(* Logix 5000 project; controller HP_SSC01 vendor 1 type 14 code 67 rev 17.7; software revision 17.01; part 10 of 15 *)
(* tags used below, declared in another part *)
   A_C3_0422 : ALIAS FOR C3_Warning.22;
   A_C3_0423 : ALIAS FOR C3_Warning.23;
   A_C3_0425 : ALIAS FOR C3_Warning.25;
   A_C3_0426 : ALIAS FOR C3_Warning.26;
   C3 : AXIS_SERVO_DRIVE;
   C3_32HourTimers : TIMER[4];
   C3_ActualPositionMOD60 : REAL;
   C3_All_DLY_OK : BOOL;
   C3_Brake_Daily_ok : BOOL;
   C3_Brake_Test_passed : BOOL;
   C3_BrakeReleaseSelected : BOOL;
   C3_BrakeTestExpireTime : DINT;
   C3_BrakeTestExpireTimeTemp : DINT;
   C3_BrakeTestFailed : BOOL;
   C3_BrakeTestMessageNumber : DINT;
   C3_BrakeTestSelected : BOOL;
   C3_BrakeTestSequence : DINT;
   C3_BrakeTestWarning : BOOL;
   C3_DistanceToEvac : REAL;
   C3_Dump_OK : BOOL;
   C3_DumpValveReleaseSelected : BOOL;
   C3_DumpValveTestExpireTime : DINT;
   C3_DumpValveTestExpireTimeTemp : DINT;
   C3_DumpValveTestSelected : BOOL;
   C3_DumpValveTestSequence : DINT;
   C3_EvacPosition : REAL;
   C3_EvacPositionMOD60 : REAL;
   C3_ExcecutePBHoldTimer : TIMER;
   C3_FaultStandard : DINT;
   C3_GoNearOnPathDelay : TIMER;
   C3_GoToEvacMAM01 : MOTION_INSTRUCTION;
   C3_GoToOnPathMAM01 : MOTION_INSTRUCTION;
   C3_GoToOnPathMAM02 : MOTION_INSTRUCTION;
   C3_Home_OK : BOOL;
   C3_Homed : BOOL;
   C3_HomeExpireTime : DINT;
   C3_HomeExpireTimeTemp : DINT;
   C3_HomeSequence : DINT;
   C3_JogForwardFastSelected : BOOL;
   C3_JogForwardSlowSelected : BOOL;
   C3_JogReverseFastSelected : BOOL;
   C3_JogReverseSlowSelected : BOOL;
   C3_LubricationMessageNumber : DINT;
   C3_LubricationOnTimer : TIMER;
   C3_LubricationOverrideSelected : BOOL;
   C3_MAFR : MOTION_INSTRUCTION;
   C3_MAG : MOTION_INSTRUCTION;
   C3_MAJDeceleration : REAL;
   C3_MAS : MOTION_INSTRUCTION;
   C3_MASR : MOTION_INSTRUCTION;
   C3_Oiler : ALIAS FOR C3_RIO_AENT:O.Data[2].1;
   C3_OIT_BrakeRelease : BOOL;
   C3_OIT_BrakeReleaseDisplay : BOOL;
   C3_OIT_BrakeTest : BOOL;
   C3_OIT_BrakeTestDisplay : BOOL;
   C3_OIT_Command : DINT;
   C3_OIT_Current : DINT;
   C3_OIT_DumpValveRelease : BOOL;
   C3_OIT_DumpValveReleaseDisplay : BOOL;
   C3_OIT_DumpValveTest : BOOL;
   C3_OIT_DumpValveTestDisplay : BOOL;
   C3_OIT_FaultsExist : BOOL;
   C3_OIT_HomeCountDown : DINT;
   C3_OIT_JogForwardFast : BOOL;
   C3_OIT_JogForwardFastDisplay : BOOL;
   C3_OIT_JogForwardSlow : BOOL;
   C3_OIT_JogForwardSlowDisplay : BOOL;
   C3_OIT_JogReverseFast : BOOL;
   C3_OIT_JogReverseFastDisplay : BOOL;
   C3_OIT_JogReverseSlow : BOOL;
   C3_OIT_JogReverseSlowDisplay : BOOL;
   C3_OIT_JogStopDisplay : BOOL;
   C3_OIT_LubricationOverride : BOOL;
   C3_OIT_LubricationOverrideDisplay : BOOL;
   C3_OIT_PathError : DINT;
   C3_OIT_PathIndicatorHigh : DINT;
   C3_OIT_PathIndicatorLow : DINT;
   C3_OIT_WarningsExist : BOOL;
   C3_OneTryToFixErrorONS : BOOL;
   C3_ONS : DINT;
   C3_RemoteBrakeAndHomeSequence : DINT;
   C3_RemoteBrakeAndHomeSequenceAlarms : DINT;
   C3_RemoteBrakeAndHomeSequenceAlarmTimer : TIMER[8];
   C3_RemoteBrakeAndHomeSequenceONS : BOOL;
   C3_RemoteBrakeTestCMD : BOOL;
   C3_RemoteDumpTestCMD : BOOL;
   C3_RemoteHomeCMD : BOOL;
   C3_RemoteScreenMessageNumber : DINT;
   C3_RemoteSequenceDelay : TIMER[4];
   C3_RevolutionCounter : COUNTER;
   C3_ServoActionStatusOnDelay : TIMER;
   C3_TargetPositionError : REAL;
   C3_TargetPositionErrorTest : REAL;
   C3_Warning : DINT;
   MasterClockCopyMAS_Stop1 : MOTION_INSTRUCTION;
   MasterClockCopyMAS_Stop2 : MOTION_INSTRUCTION;
   MasterClockLocal : AXIS_VIRTUAL;
   RCS_CMD_Auto_TON : TIMER;
   RCS_MasterClockLocalTagetDegrees : REAL;
   S_C3_FaultReset : BOOL;
   S_C3_FaultSafety : DINT;
   S_C3_ModeLocal : BOOL;
   S_C3_ModeRemote : BOOL;
   S_C3_MSTOP_InputOK : BOOL;
   S_C3_NearOnPath : BOOL;
   S_C3_NearOnPathHi : DINT;
   S_C3_NearOnPathLow : DINT;
   S_C3_OffPath : BOOL;
   S_C3_OnPath : BOOL;
   S_C3_PathError : DINT;
   S_RCS_MotionCMD_BrakeTest : BOOL;
   S_RCS_MotionCMD_Evac : BOOL;
   S_RCS_MotionCMD_GoNearOnPath : BOOL;
(* Carousel3, continued *)

ROUTINE C345_Lubrication   (* ladder *)
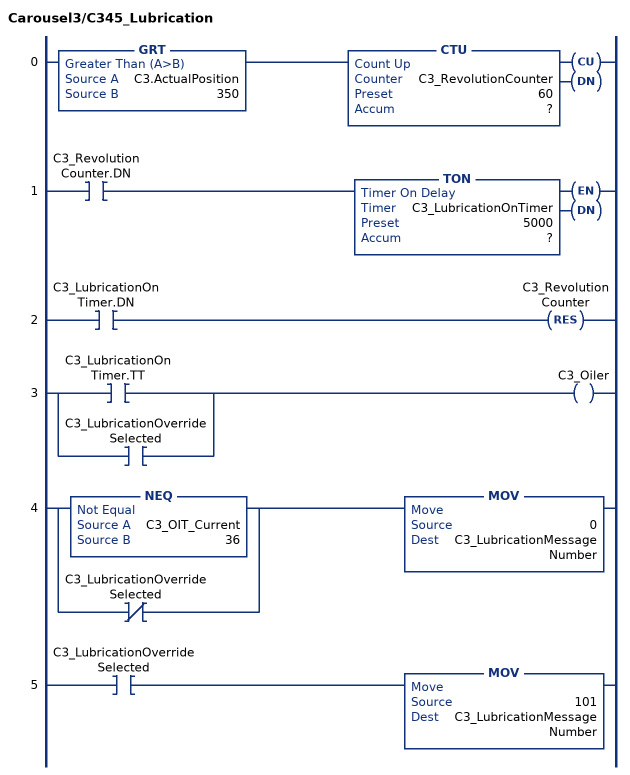
   0: GRT(C3.ActualPosition,350)CTU(C3_RevolutionCounter,?,?);
   1: XIC(C3_RevolutionCounter.DN)TON(C3_LubricationOnTimer,?,?);
   2: XIC(C3_LubricationOnTimer.DN)RES(C3_RevolutionCounter);
   3: [XIC(C3_LubricationOnTimer.TT) ,XIC(C3_LubricationOverrideSelected) ]OTE(C3_Oiler);
   4: [NEQ(C3_OIT_Current,36) ,XIO(C3_LubricationOverrideSelected) ]MOV(0,C3_LubricationMessageNumber);
   5: XIC(C3_LubricationOverrideSelected)MOV(101,C3_LubricationMessageNumber);
END_ROUTINE

ROUTINE C350_OIT   (* ladder *)
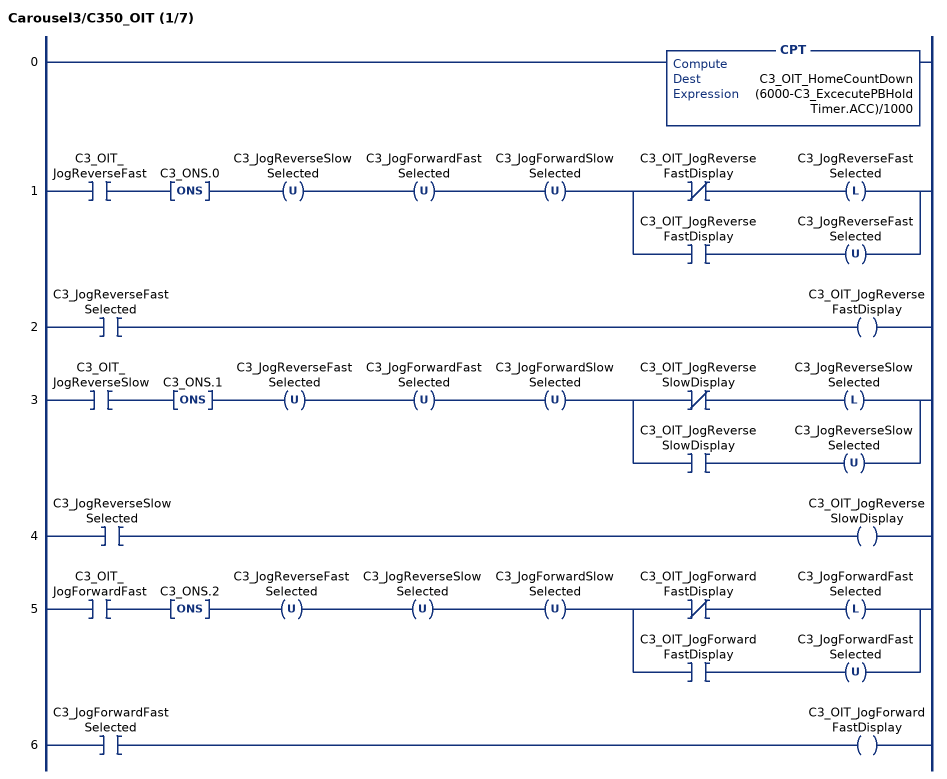
   0: CPT(C3_OIT_HomeCountDown,(6000-C3_ExcecutePBHoldTimer.ACC)/1000);
   1: XIC(C3_OIT_JogReverseFast)ONS(C3_ONS.0)OTU(C3_JogReverseSlowSelected)OTU(C3_JogForwardFastSelected)OTU(C3_JogForwardSlowSelected)[XIO(C3_OIT_JogReverseFastDisplay) OTL(C3_JogReverseFastSelected) ,XIC(C3_OIT_JogReverseFastDisplay) OTU(C3_JogReverseFastSelected) ];
   2: XIC(C3_JogReverseFastSelected)OTE(C3_OIT_JogReverseFastDisplay);
   3: XIC(C3_OIT_JogReverseSlow)ONS(C3_ONS.1)OTU(C3_JogReverseFastSelected)OTU(C3_JogForwardFastSelected)OTU(C3_JogForwardSlowSelected)[XIO(C3_OIT_JogReverseSlowDisplay) OTL(C3_JogReverseSlowSelected) ,XIC(C3_OIT_JogReverseSlowDisplay) OTU(C3_JogReverseSlowSelected) ];
   4: XIC(C3_JogReverseSlowSelected)OTE(C3_OIT_JogReverseSlowDisplay);
   5: XIC(C3_OIT_JogForwardFast)ONS(C3_ONS.2)OTU(C3_JogReverseFastSelected)OTU(C3_JogReverseSlowSelected)OTU(C3_JogForwardSlowSelected)[XIO(C3_OIT_JogForwardFastDisplay) OTL(C3_JogForwardFastSelected) ,XIC(C3_OIT_JogForwardFastDisplay) OTU(C3_JogForwardFastSelected) ];
   6: XIC(C3_JogForwardFastSelected)OTE(C3_OIT_JogForwardFastDisplay);
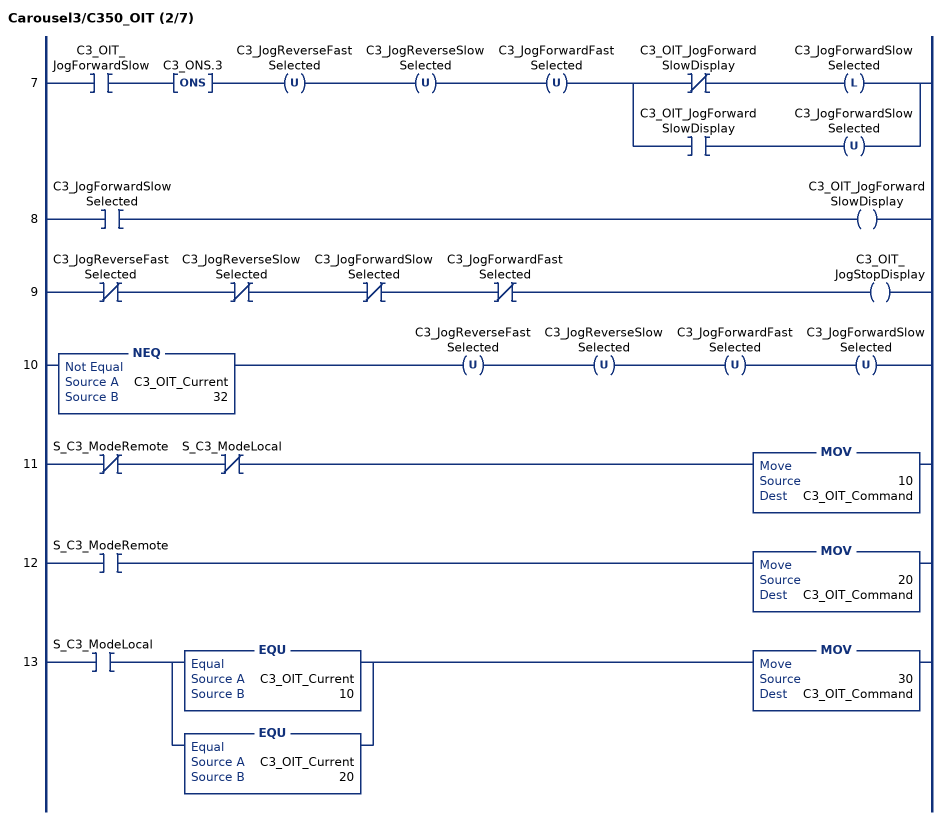
   7: XIC(C3_OIT_JogForwardSlow)ONS(C3_ONS.3)OTU(C3_JogReverseFastSelected)OTU(C3_JogReverseSlowSelected)OTU(C3_JogForwardFastSelected)[XIO(C3_OIT_JogForwardSlowDisplay) OTL(C3_JogForwardSlowSelected) ,XIC(C3_OIT_JogForwardSlowDisplay) OTU(C3_JogForwardSlowSelected) ];
   8: XIC(C3_JogForwardSlowSelected)OTE(C3_OIT_JogForwardSlowDisplay);
   9: XIO(C3_JogReverseFastSelected)XIO(C3_JogReverseSlowSelected)XIO(C3_JogForwardSlowSelected)XIO(C3_JogForwardFastSelected)OTE(C3_OIT_JogStopDisplay);
   10: NEQ(C3_OIT_Current,32)OTU(C3_JogReverseFastSelected)OTU(C3_JogReverseSlowSelected)OTU(C3_JogForwardFastSelected)OTU(C3_JogForwardSlowSelected);
   11: XIO(S_C3_ModeRemote)XIO(S_C3_ModeLocal)MOV(10,C3_OIT_Command);
   12: XIC(S_C3_ModeRemote)MOV(20,C3_OIT_Command);
   13: XIC(S_C3_ModeLocal)[EQU(C3_OIT_Current,10) ,EQU(C3_OIT_Current,20) ]MOV(30,C3_OIT_Command);
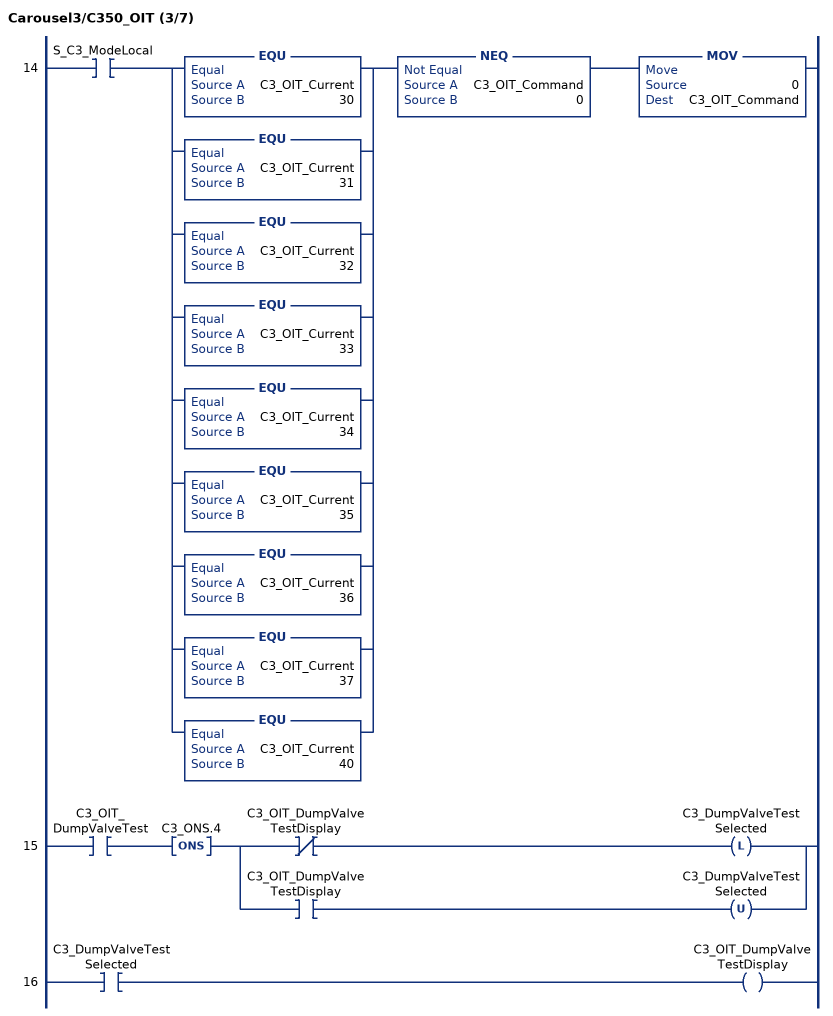
   14: XIC(S_C3_ModeLocal)[EQU(C3_OIT_Current,30) ,EQU(C3_OIT_Current,31) ,EQU(C3_OIT_Current,32) ,EQU(C3_OIT_Current,33) ,EQU(C3_OIT_Current,34) ,EQU(C3_OIT_Current,35) ,EQU(C3_OIT_Current,36) ,EQU(C3_OIT_Current,37) ,EQU(C3_OIT_Current,40) ]NEQ(C3_OIT_Command,0)MOV(0,C3_OIT_Command);
   15: XIC(C3_OIT_DumpValveTest)ONS(C3_ONS.4)[XIO(C3_OIT_DumpValveTestDisplay) OTL(C3_DumpValveTestSelected) ,XIC(C3_OIT_DumpValveTestDisplay) OTU(C3_DumpValveTestSelected) ];
   16: XIC(C3_DumpValveTestSelected)OTE(C3_OIT_DumpValveTestDisplay);
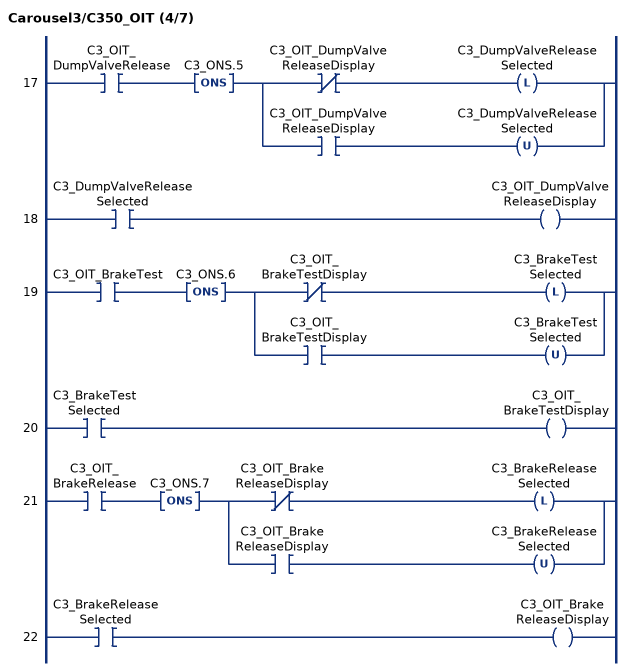
   17: XIC(C3_OIT_DumpValveRelease)ONS(C3_ONS.5)[XIO(C3_OIT_DumpValveReleaseDisplay) OTL(C3_DumpValveReleaseSelected) ,XIC(C3_OIT_DumpValveReleaseDisplay) OTU(C3_DumpValveReleaseSelected) ];
   18: XIC(C3_DumpValveReleaseSelected)OTE(C3_OIT_DumpValveReleaseDisplay);
   19: XIC(C3_OIT_BrakeTest)ONS(C3_ONS.6)[XIO(C3_OIT_BrakeTestDisplay) OTL(C3_BrakeTestSelected) ,XIC(C3_OIT_BrakeTestDisplay) OTU(C3_BrakeTestSelected) ];
   20: XIC(C3_BrakeTestSelected)OTE(C3_OIT_BrakeTestDisplay);
   21: XIC(C3_OIT_BrakeRelease)ONS(C3_ONS.7)[XIO(C3_OIT_BrakeReleaseDisplay) OTL(C3_BrakeReleaseSelected) ,XIC(C3_OIT_BrakeReleaseDisplay) OTU(C3_BrakeReleaseSelected) ];
   22: XIC(C3_BrakeReleaseSelected)OTE(C3_OIT_BrakeReleaseDisplay);
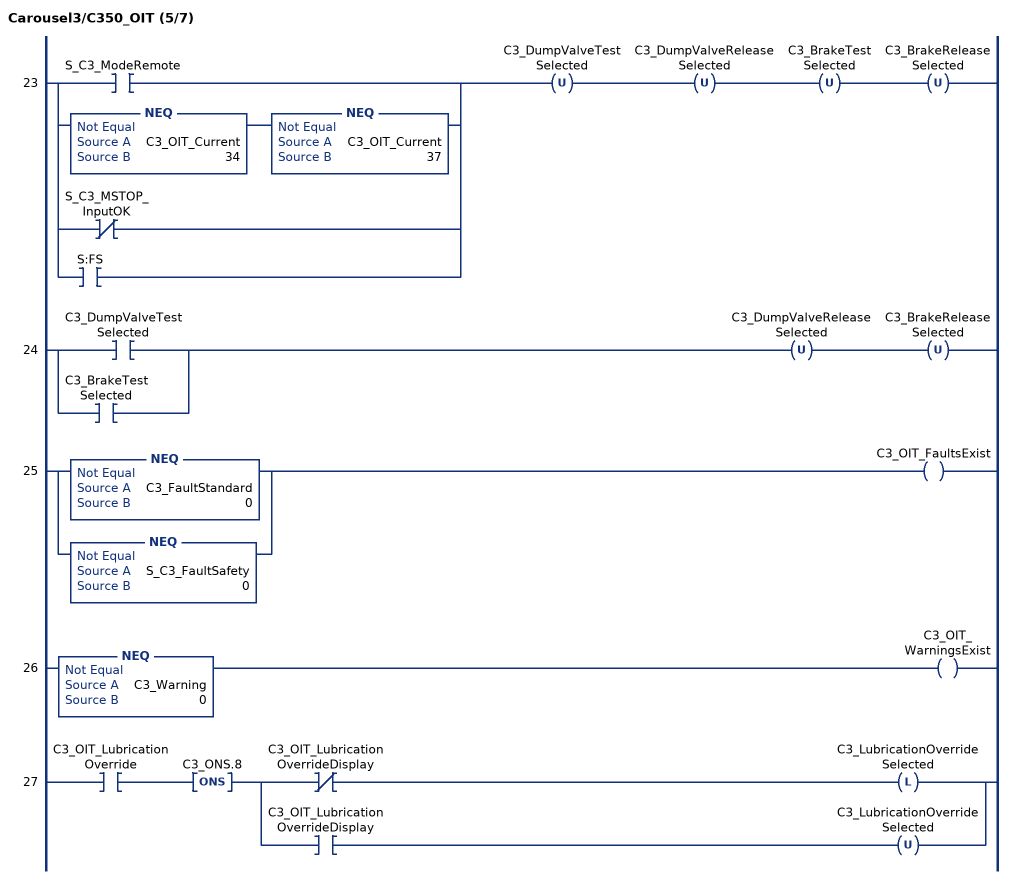
   23: [XIC(S_C3_ModeRemote) ,NEQ(C3_OIT_Current,34) NEQ(C3_OIT_Current,37) ,XIO(S_C3_MSTOP_InputOK) ,XIC(S:FS) ]OTU(C3_DumpValveTestSelected)OTU(C3_DumpValveReleaseSelected)OTU(C3_BrakeTestSelected)OTU(C3_BrakeReleaseSelected);
   24: [XIC(C3_DumpValveTestSelected) ,XIC(C3_BrakeTestSelected) ]OTU(C3_DumpValveReleaseSelected)OTU(C3_BrakeReleaseSelected);
   25: [NEQ(C3_FaultStandard,0) ,NEQ(S_C3_FaultSafety,0) ]OTE(C3_OIT_FaultsExist);
   26: NEQ(C3_Warning,0)OTE(C3_OIT_WarningsExist);
   27: XIC(C3_OIT_LubricationOverride)ONS(C3_ONS.8)[XIO(C3_OIT_LubricationOverrideDisplay) OTL(C3_LubricationOverrideSelected) ,XIC(C3_OIT_LubricationOverrideDisplay) OTU(C3_LubricationOverrideSelected) ];
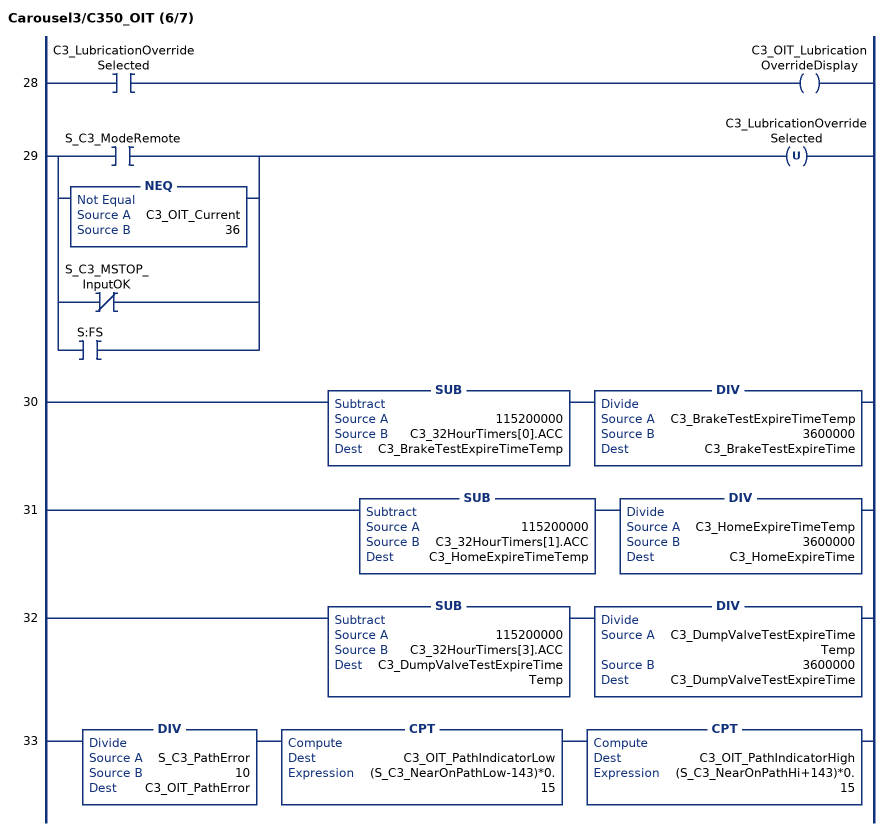
   28: XIC(C3_LubricationOverrideSelected)OTE(C3_OIT_LubricationOverrideDisplay);
   29: [XIC(S_C3_ModeRemote) ,NEQ(C3_OIT_Current,36) ,XIO(S_C3_MSTOP_InputOK) ,XIC(S:FS) ]OTU(C3_LubricationOverrideSelected);
   30: SUB(115200000,C3_32HourTimers[0].ACC,C3_BrakeTestExpireTimeTemp)DIV(C3_BrakeTestExpireTimeTemp,3600000,C3_BrakeTestExpireTime);
   31: SUB(115200000,C3_32HourTimers[1].ACC,C3_HomeExpireTimeTemp)DIV(C3_HomeExpireTimeTemp,3600000,C3_HomeExpireTime);
   32: SUB(115200000,C3_32HourTimers[3].ACC,C3_DumpValveTestExpireTimeTemp)DIV(C3_DumpValveTestExpireTimeTemp,3600000,C3_DumpValveTestExpireTime);
   33: DIV(S_C3_PathError,10,C3_OIT_PathError)CPT(C3_OIT_PathIndicatorLow,(S_C3_NearOnPathLow-143)*0.15)CPT(C3_OIT_PathIndicatorHigh,(S_C3_NearOnPathHi+143)*0.15);
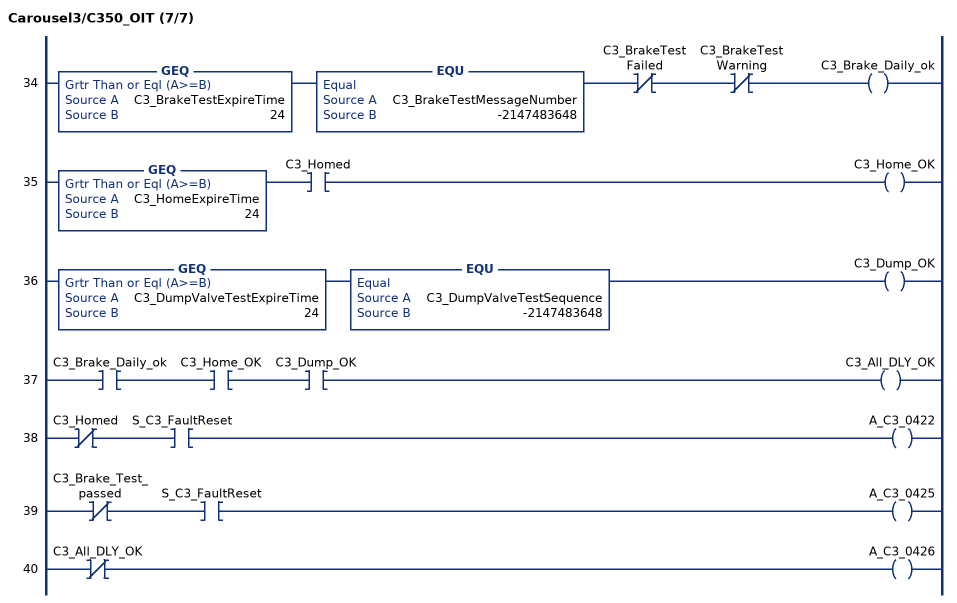
   34: GEQ(C3_BrakeTestExpireTime,24)EQU(C3_BrakeTestMessageNumber,-2147483648)XIO(C3_BrakeTestFailed)XIO(C3_BrakeTestWarning)OTE(C3_Brake_Daily_ok);
   35: GEQ(C3_HomeExpireTime,24)XIC(C3_Homed)OTE(C3_Home_OK);
   36: GEQ(C3_DumpValveTestExpireTime,24)EQU(C3_DumpValveTestSequence,-2147483648)OTE(C3_Dump_OK);
   37: XIC(C3_Brake_Daily_ok)XIC(C3_Home_OK)XIC(C3_Dump_OK)OTE(C3_All_DLY_OK);
   38: XIO(C3_Homed)XIC(S_C3_FaultReset)OTE(A_C3_0422);
   39: XIO(C3_Brake_Test_passed)XIC(S_C3_FaultReset)OTE(A_C3_0425);
   40: XIO(C3_All_DLY_OK)OTE(A_C3_0426);
END_ROUTINE

ROUTINE C355_Remote   (* ladder *)
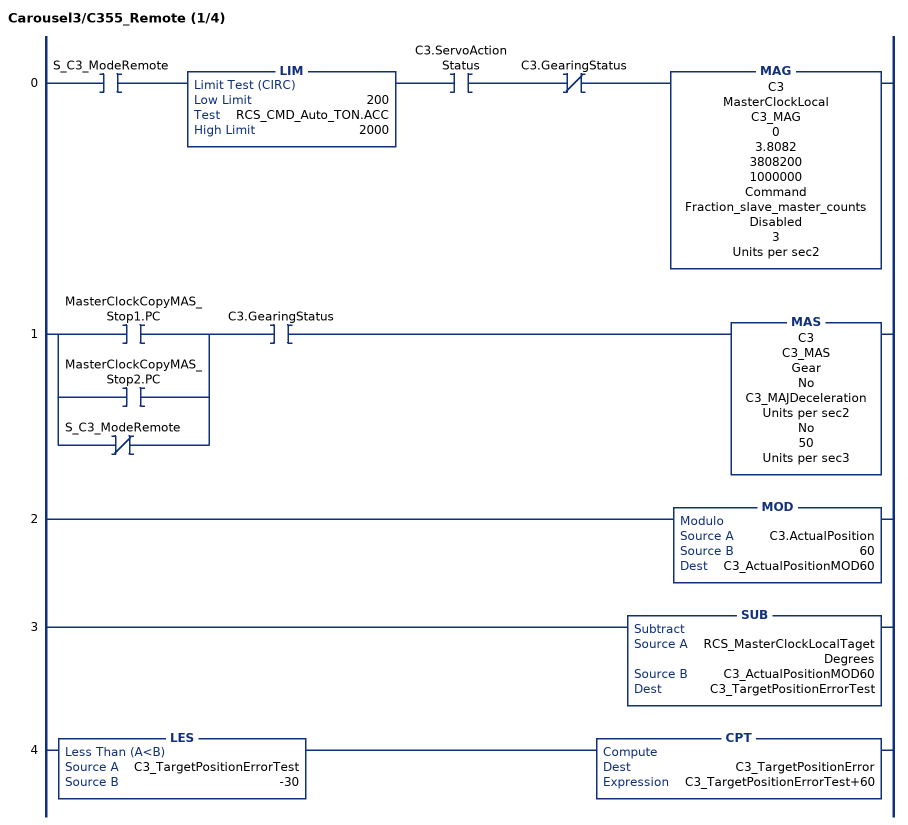
   0: XIC(S_C3_ModeRemote)LIM(200,RCS_CMD_Auto_TON.ACC,2000)XIC(C3.ServoActionStatus)XIO(C3.GearingStatus)MAG(C3,MasterClockLocal,C3_MAG,0,3.8082,3808200,1000000,Command,Fraction_slave_master_counts,Disabled,3,Units per sec2);
   1: [XIC(MasterClockCopyMAS_Stop1.PC) ,XIC(MasterClockCopyMAS_Stop2.PC) ,XIO(S_C3_ModeRemote) ]XIC(C3.GearingStatus)MAS(C3,C3_MAS,Gear,No,C3_MAJDeceleration,Units per sec2,No,50,Units per sec3);
   2: MOD(C3.ActualPosition,60,C3_ActualPositionMOD60);
   3: SUB(RCS_MasterClockLocalTagetDegrees,C3_ActualPositionMOD60,C3_TargetPositionErrorTest);
   4: LES(C3_TargetPositionErrorTest,-30)CPT(C3_TargetPositionError,C3_TargetPositionErrorTest+60);
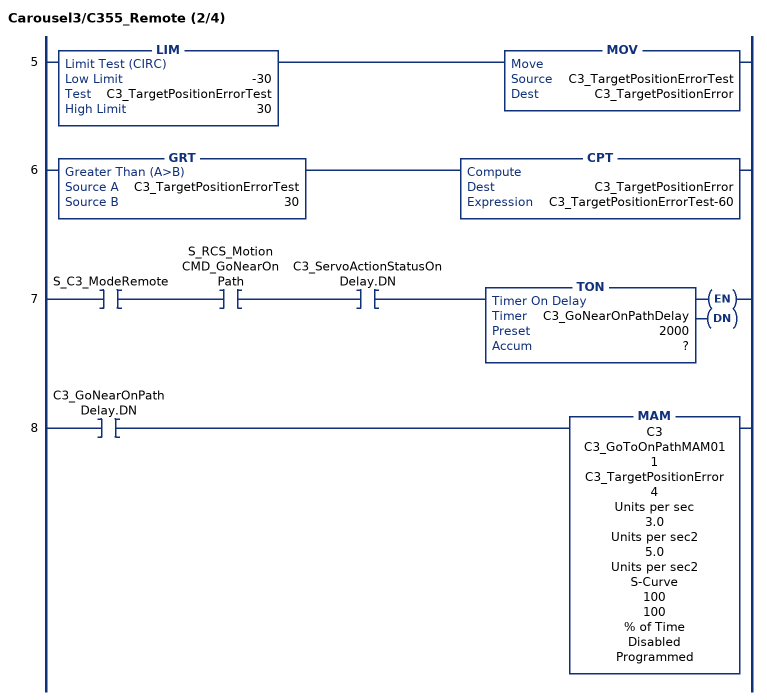
   5: LIM(-30,C3_TargetPositionErrorTest,30)MOV(C3_TargetPositionErrorTest,C3_TargetPositionError);
   6: GRT(C3_TargetPositionErrorTest,30)CPT(C3_TargetPositionError,C3_TargetPositionErrorTest-60);
   7: XIC(S_C3_ModeRemote)XIC(S_RCS_MotionCMD_GoNearOnPath)XIC(C3_ServoActionStatusOnDelay.DN)TON(C3_GoNearOnPathDelay,?,?);
   8: XIC(C3_GoNearOnPathDelay.DN)MAM(C3,C3_GoToOnPathMAM01,1,C3_TargetPositionError,4,Units per sec,3.0,Units per sec2,5.0,Units per sec2,S-Curve,100,100,% of Time,Disabled,Programmed);
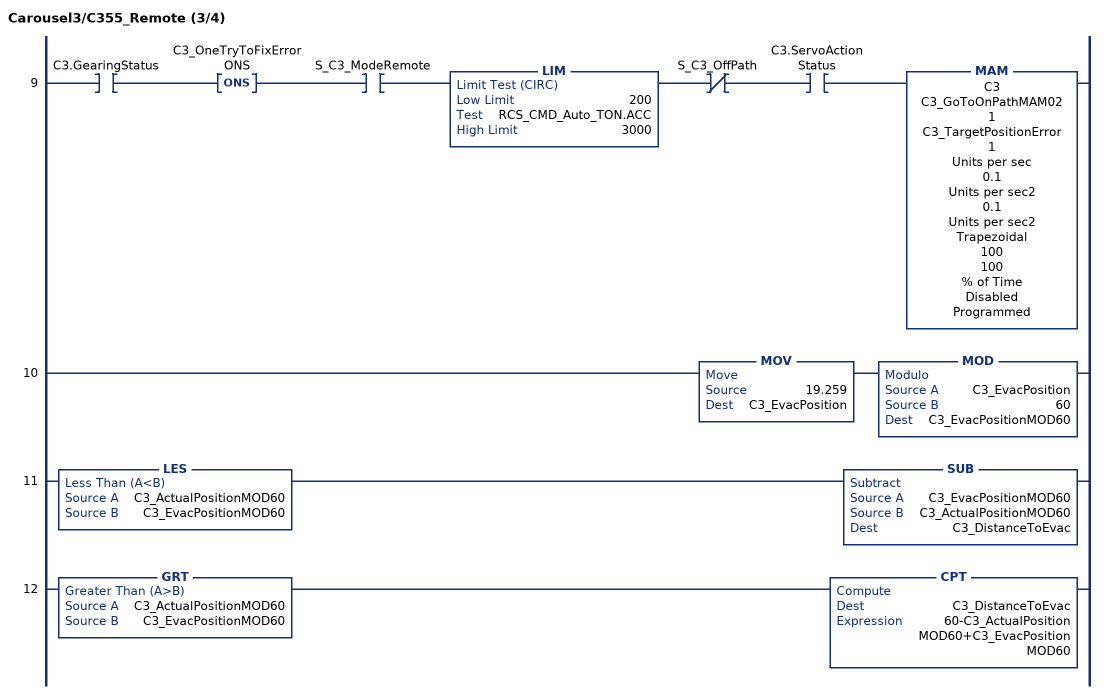
   9: XIC(C3.GearingStatus)ONS(C3_OneTryToFixErrorONS)XIC(S_C3_ModeRemote)LIM(200,RCS_CMD_Auto_TON.ACC,3000)XIO(S_C3_OffPath)XIC(C3.ServoActionStatus)MAM(C3,C3_GoToOnPathMAM02,1,C3_TargetPositionError,1,Units per sec,0.1,Units per sec2,0.1,Units per sec2,Trapezoidal,100,100,% of Time,Disabled,Programmed);
   10: MOV(19.259,C3_EvacPosition)MOD(C3_EvacPosition,60,C3_EvacPositionMOD60);
   11: LES(C3_ActualPositionMOD60,C3_EvacPositionMOD60)SUB(C3_EvacPositionMOD60,C3_ActualPositionMOD60,C3_DistanceToEvac);
   12: GRT(C3_ActualPositionMOD60,C3_EvacPositionMOD60)CPT(C3_DistanceToEvac,60-C3_ActualPositionMOD60+C3_EvacPositionMOD60);
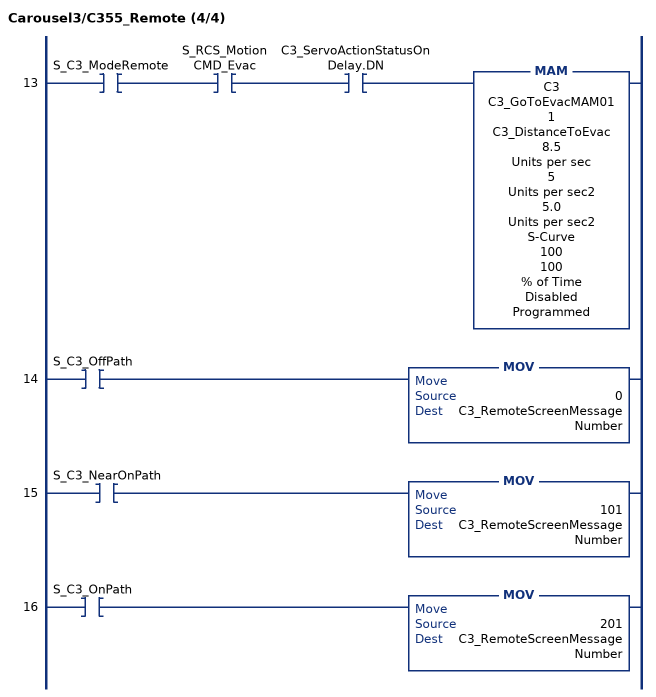
   13: XIC(S_C3_ModeRemote)XIC(S_RCS_MotionCMD_Evac)XIC(C3_ServoActionStatusOnDelay.DN)MAM(C3,C3_GoToEvacMAM01,1,C3_DistanceToEvac,8.5,Units per sec,5,Units per sec2,5.0,Units per sec2,S-Curve,100,100,% of Time,Disabled,Programmed);
   14: XIC(S_C3_OffPath)MOV(0,C3_RemoteScreenMessageNumber);
   15: XIC(S_C3_NearOnPath)MOV(101,C3_RemoteScreenMessageNumber);
   16: XIC(S_C3_OnPath)MOV(201,C3_RemoteScreenMessageNumber);
END_ROUTINE

ROUTINE C360_RemoteBrakeAndHome   (* ladder *)
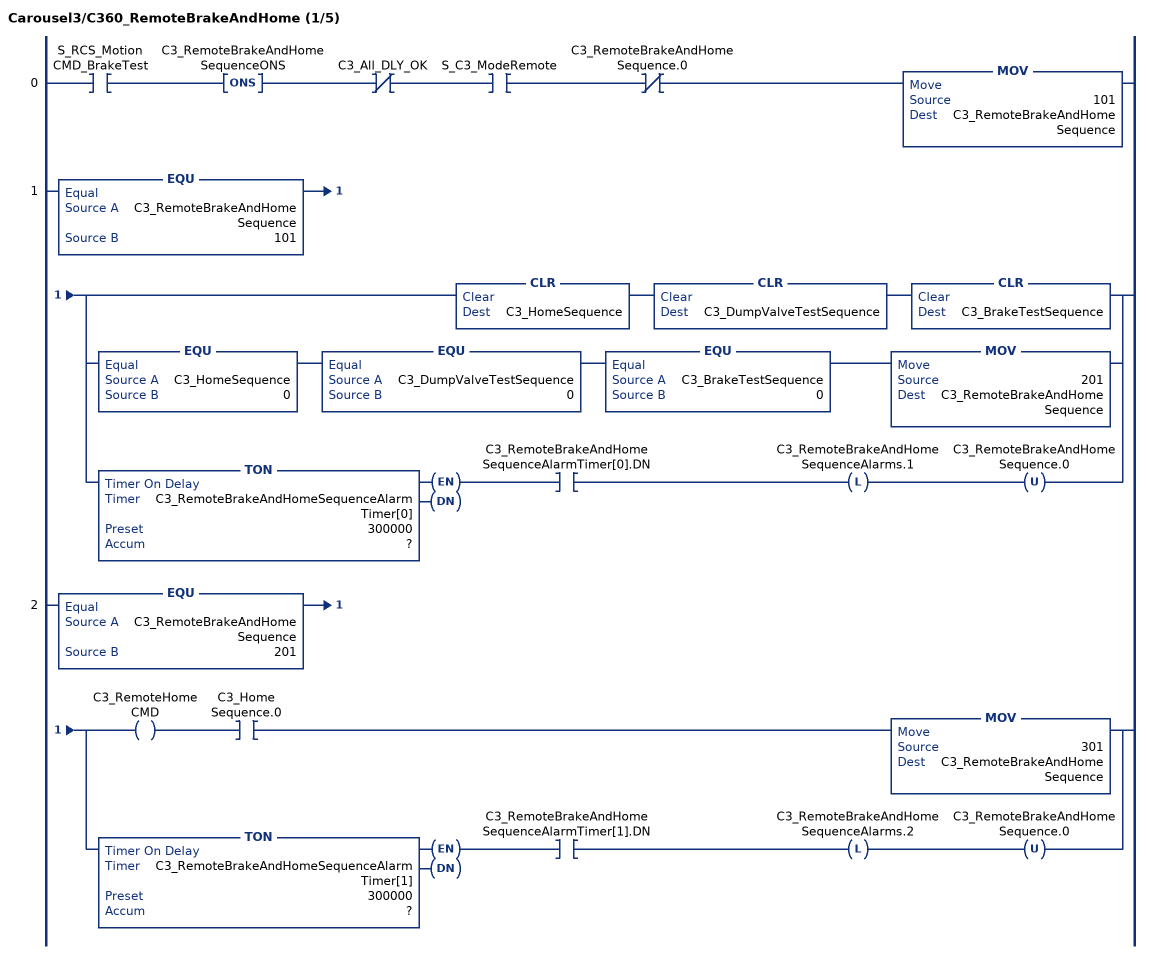
   0: XIC(S_RCS_MotionCMD_BrakeTest)ONS(C3_RemoteBrakeAndHomeSequenceONS)XIO(C3_All_DLY_OK)XIC(S_C3_ModeRemote)XIO(C3_RemoteBrakeAndHomeSequence.0)MOV(101,C3_RemoteBrakeAndHomeSequence);
   1: EQU(C3_RemoteBrakeAndHomeSequence,101)[CLR(C3_HomeSequence) CLR(C3_DumpValveTestSequence) CLR(C3_BrakeTestSequence) ,EQU(C3_HomeSequence,0) EQU(C3_DumpValveTestSequence,0) EQU(C3_BrakeTestSequence,0) MOV(201,C3_RemoteBrakeAndHomeSequence) ,TON(C3_RemoteBrakeAndHomeSequenceAlarmTimer[0],?,?) XIC(C3_RemoteBrakeAndHomeSequenceAlarmTimer[0].DN) OTL(C3_RemoteBrakeAndHomeSequenceAlarms.1) OTU(C3_RemoteBrakeAndHomeSequence.0) ];
   2: EQU(C3_RemoteBrakeAndHomeSequence,201)[OTE(C3_RemoteHomeCMD) XIC(C3_HomeSequence.0) MOV(301,C3_RemoteBrakeAndHomeSequence) ,TON(C3_RemoteBrakeAndHomeSequenceAlarmTimer[1],?,?) XIC(C3_RemoteBrakeAndHomeSequenceAlarmTimer[1].DN) OTL(C3_RemoteBrakeAndHomeSequenceAlarms.2) OTU(C3_RemoteBrakeAndHomeSequence.0) ];
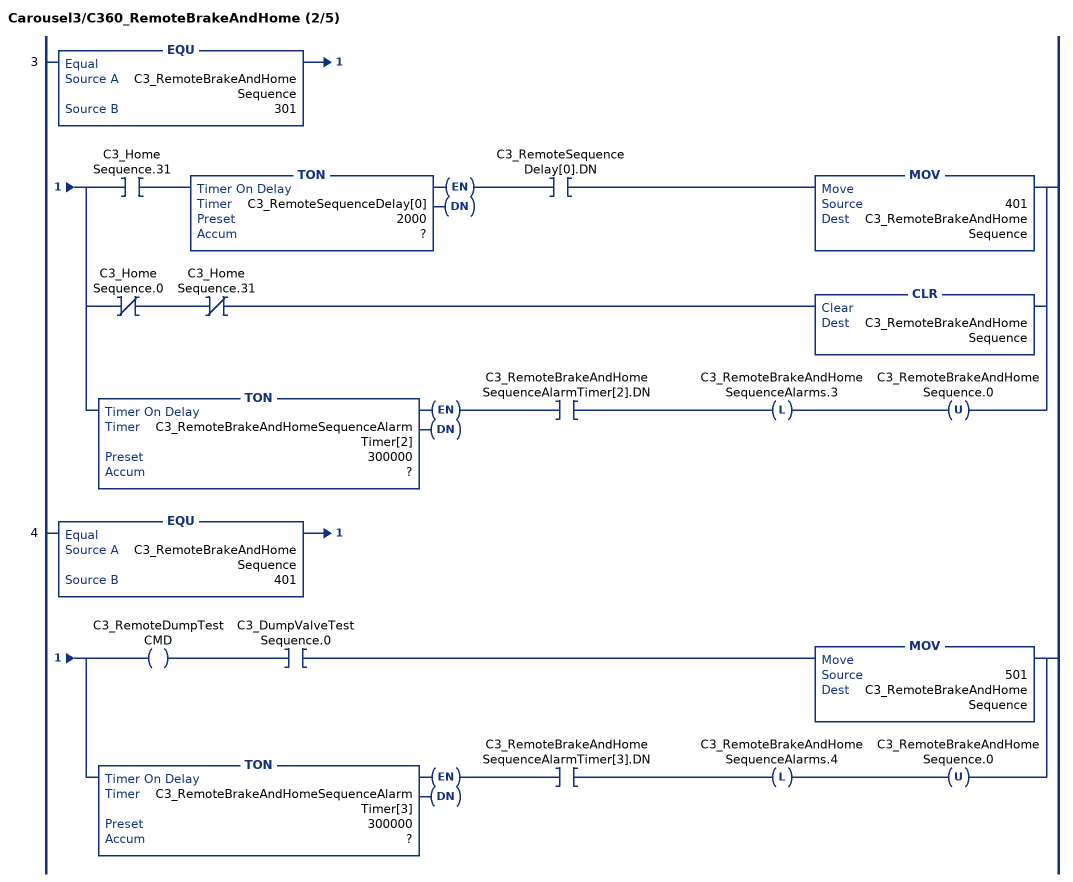
   3: EQU(C3_RemoteBrakeAndHomeSequence,301)[XIC(C3_HomeSequence.31) TON(C3_RemoteSequenceDelay[0],?,?) XIC(C3_RemoteSequenceDelay[0].DN) MOV(401,C3_RemoteBrakeAndHomeSequence) ,XIO(C3_HomeSequence.0) XIO(C3_HomeSequence.31) CLR(C3_RemoteBrakeAndHomeSequence) ,TON(C3_RemoteBrakeAndHomeSequenceAlarmTimer[2],?,?) XIC(C3_RemoteBrakeAndHomeSequenceAlarmTimer[2].DN) OTL(C3_RemoteBrakeAndHomeSequenceAlarms.3) OTU(C3_RemoteBrakeAndHomeSequence.0) ];
   4: EQU(C3_RemoteBrakeAndHomeSequence,401)[OTE(C3_RemoteDumpTestCMD) XIC(C3_DumpValveTestSequence.0) MOV(501,C3_RemoteBrakeAndHomeSequence) ,TON(C3_RemoteBrakeAndHomeSequenceAlarmTimer[3],?,?) XIC(C3_RemoteBrakeAndHomeSequenceAlarmTimer[3].DN) OTL(C3_RemoteBrakeAndHomeSequenceAlarms.4) OTU(C3_RemoteBrakeAndHomeSequence.0) ];
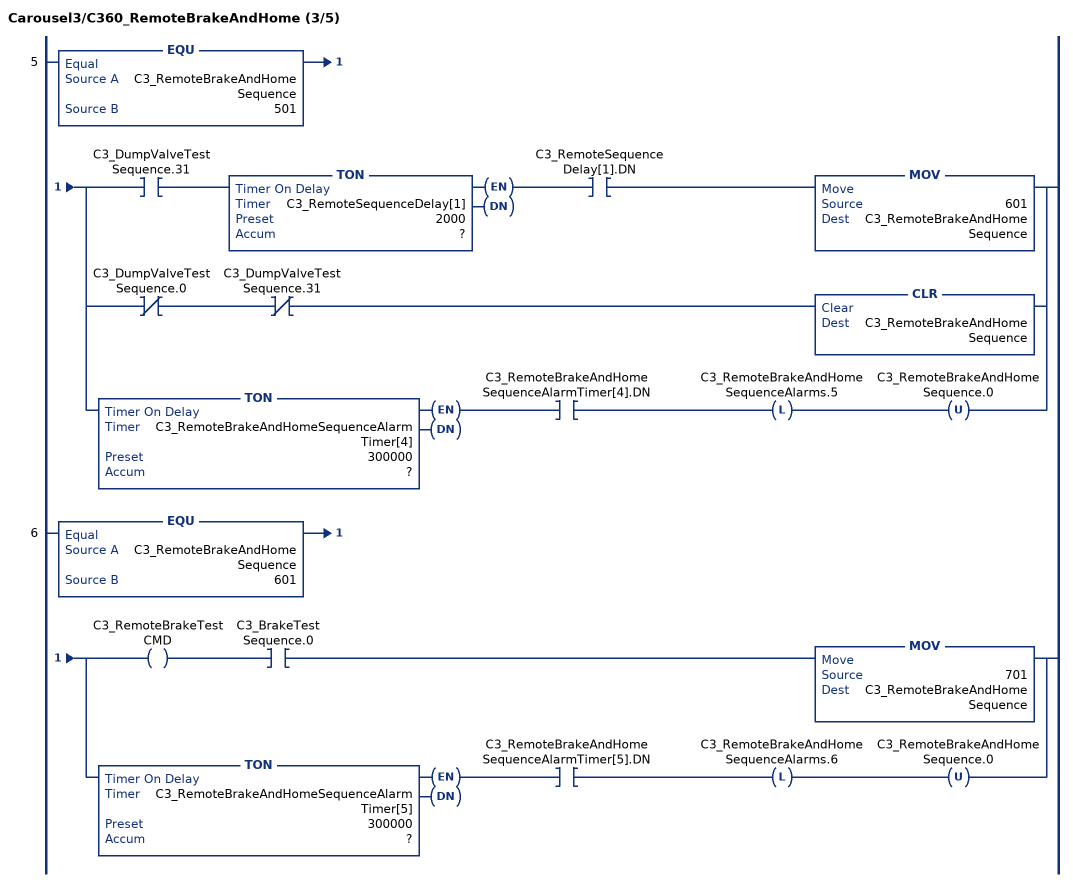
   5: EQU(C3_RemoteBrakeAndHomeSequence,501)[XIC(C3_DumpValveTestSequence.31) TON(C3_RemoteSequenceDelay[1],?,?) XIC(C3_RemoteSequenceDelay[1].DN) MOV(601,C3_RemoteBrakeAndHomeSequence) ,XIO(C3_DumpValveTestSequence.0) XIO(C3_DumpValveTestSequence.31) CLR(C3_RemoteBrakeAndHomeSequence) ,TON(C3_RemoteBrakeAndHomeSequenceAlarmTimer[4],?,?) XIC(C3_RemoteBrakeAndHomeSequenceAlarmTimer[4].DN) OTL(C3_RemoteBrakeAndHomeSequenceAlarms.5) OTU(C3_RemoteBrakeAndHomeSequence.0) ];
   6: EQU(C3_RemoteBrakeAndHomeSequence,601)[OTE(C3_RemoteBrakeTestCMD) XIC(C3_BrakeTestSequence.0) MOV(701,C3_RemoteBrakeAndHomeSequence) ,TON(C3_RemoteBrakeAndHomeSequenceAlarmTimer[5],?,?) XIC(C3_RemoteBrakeAndHomeSequenceAlarmTimer[5].DN) OTL(C3_RemoteBrakeAndHomeSequenceAlarms.6) OTU(C3_RemoteBrakeAndHomeSequence.0) ];
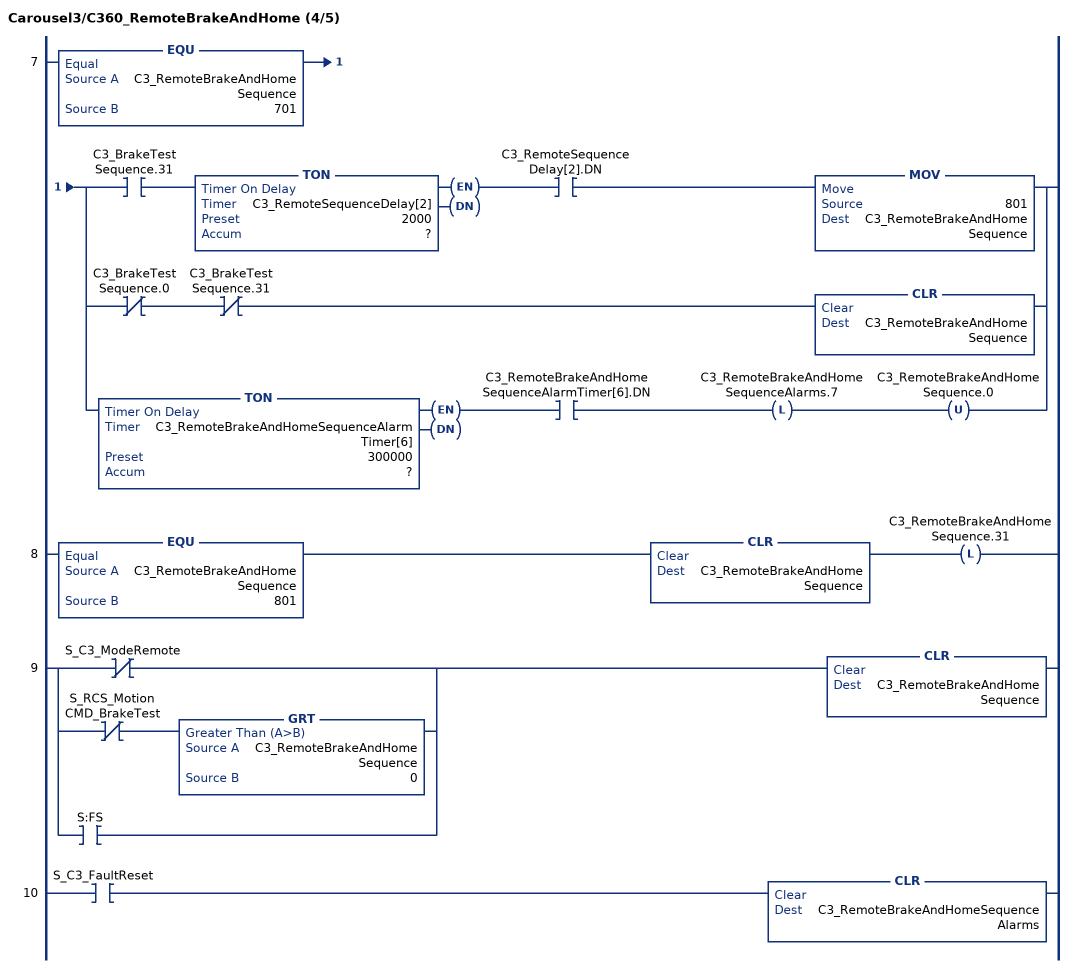
   7: EQU(C3_RemoteBrakeAndHomeSequence,701)[XIC(C3_BrakeTestSequence.31) TON(C3_RemoteSequenceDelay[2],?,?) XIC(C3_RemoteSequenceDelay[2].DN) MOV(801,C3_RemoteBrakeAndHomeSequence) ,XIO(C3_BrakeTestSequence.0) XIO(C3_BrakeTestSequence.31) CLR(C3_RemoteBrakeAndHomeSequence) ,TON(C3_RemoteBrakeAndHomeSequenceAlarmTimer[6],?,?) XIC(C3_RemoteBrakeAndHomeSequenceAlarmTimer[6].DN) OTL(C3_RemoteBrakeAndHomeSequenceAlarms.7) OTU(C3_RemoteBrakeAndHomeSequence.0) ];
   8: EQU(C3_RemoteBrakeAndHomeSequence,801)CLR(C3_RemoteBrakeAndHomeSequence)OTL(C3_RemoteBrakeAndHomeSequence.31);
   9: [XIO(S_C3_ModeRemote) ,XIO(S_RCS_MotionCMD_BrakeTest) GRT(C3_RemoteBrakeAndHomeSequence,0) ,XIC(S:FS) ]CLR(C3_RemoteBrakeAndHomeSequence);
   10: XIC(S_C3_FaultReset)CLR(C3_RemoteBrakeAndHomeSequenceAlarms);
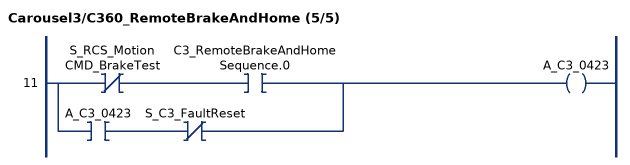
   11: [XIO(S_RCS_MotionCMD_BrakeTest) XIC(C3_RemoteBrakeAndHomeSequence.0) ,XIC(A_C3_0423) XIO(S_C3_FaultReset) ]OTE(A_C3_0423);
END_ROUTINE

ROUTINE C365_Reset   (* ladder *)
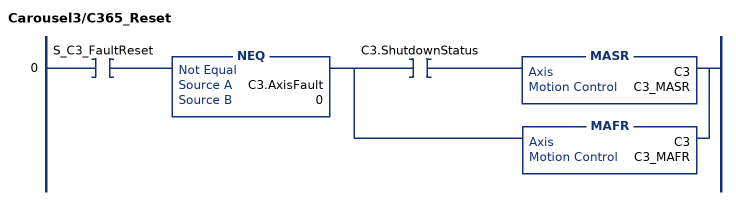
   0: XIC(S_C3_FaultReset)NEQ(C3.AxisFault,0)[XIC(C3.ShutdownStatus) MASR(C3,C3_MASR) ,MAFR(C3,C3_MAFR) ];
END_ROUTINE
END_PROGRAM
